DATA_BLOCK "InstCalculator"
{ S7_Optimized_Access := 'TRUE' }
VERSION : 0.1
NON_RETAIN
"Calculator"

BEGIN

END_DATA_BLOCK

